// TIA Portal V18 export
FUNCTION_BLOCK "FB_Tower_4Lamp"   // FB5050, LAD
{ S7_Optimized_Access := 'TRUE' }
VERSION : 0.1
// stored: AutoNumber false, IsIECCheckEnabled false, IsRetainMemResEnabled false, MemoryReserve 100, SetENOAutomatically false, UDAEnableTagReadback false
   VAR_INPUT
      iReady : Bool;   // 系统OK
      iManual_Mode : Bool;
      iAuto_Mode : Bool;
      iAuto_Running : Bool;   // 自动运行信号
      iCheck_Mode : Bool;
      iIdle : Bool;   // 自动运行中空闲信号
      iWarning : Bool;
      iFault : Bool;
      "i0.5s_Pulse" : Bool;   // 0.5S脉冲
      i1s_Pulse : Bool;   // 1S脉冲
      i2s_Pulse : Bool;   // 2S脉冲
      iResetButton : Bool;   // 复位按钮
      "iE-StopButtonOK" : Bool;   // 急停按钮未按下
      iSafetyGateClosed : Bool;   // 安全门关闭信号
      iSafetyGateRelayOK : Bool;   // 安全门继电器输出OK
      iPowerOn : Bool;   // 系统上电信号
      iMachineHomePos : Bool;   // 所有设备在原始位
      iWorkAreaLightButton : Bool;   // HMI工作区域照明按钮
      iTest_Lamp : Bool;   // 灯测试按钮
   END_VAR
   VAR_OUTPUT
      oRed_Lamp : Bool;   // 塔灯-红色
      oYellow_Lamp : Bool;   // 塔灯-黄色
      oGreen_Lamp : Bool;   // 塔灯-绿色
      oBlue_Lamp : Bool;   // 塔灯-蓝色 1.蓝灯常亮表示设备在原位;2.蓝灯闪烁表示工位缺料等待上料
      oBuzzer : Bool;   // 塔灯-蜂鸣器
      oPowerOn : Bool;   // 系统上电指示灯
      oResetLamp : Bool;   // 复位按钮指示灯
      oWorkArea1_LightingOn : Bool;   // 工作区域1 照明打开
      oWorkArea2_LightingOn : Bool;   // 工作区域2 照明打开
      oWorkArea3_LightingOn : Bool;   // 工作区域3 照明打开
   END_VAR
   VAR_IN_OUT
      ioStationWaitingLoadPart : Bool;   // 工位等待工位上料
      ioBuzzerON : Bool;   // 蜂鸣器屏蔽开关
      ioBuzzerSetVal : Int;   // 蜂鸣器鸣叫设定值
   END_VAR
   VAR
      TON : Array[0..10] of TON_TIME;
      sRed_Lamp { S7_SetPoint := 'True'} : Bool;
      sResetButtonPressed : Bool;   // 复位按钮已按下
      sBuzzerOnCurrentVal : Int;   // 蜂鸣器鸣叫实际值
      P_TRIG : Array[0..10] of Bool;
      N_TRIG : Array[0..10] of Bool;
   END_VAR
   VAR_TEMP   // added for the SCL form of the ladder/FBD networks
      _w1 : Bool;
      _w2 : Bool;
      _w3 : Bool;
      _w4 : Bool;
      _w5 : Bool;
      _w6 : Bool;
   END_VAR
BEGIN

REGION Network 1: 塔灯-红色 / TowerLamp_Red
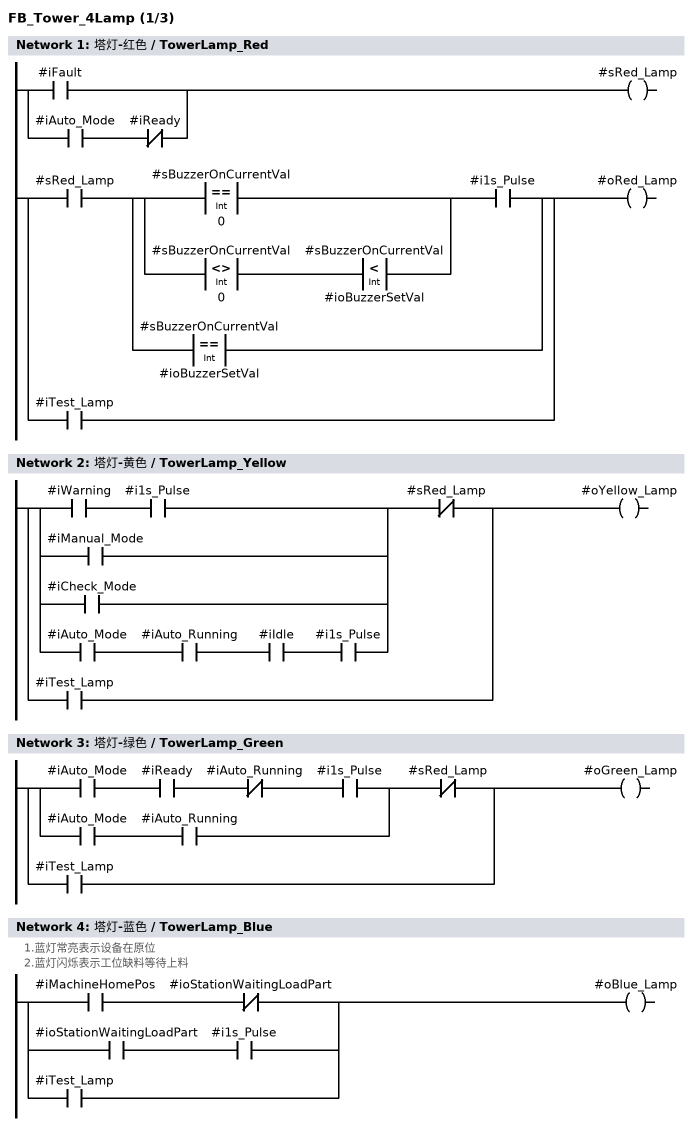
   RUNG wire#powerrail
      Contact( #iFault )
      wire#w1
      Coil( #sRed_Lamp )
   END_RUNG
   RUNG wire#powerrail
      Contact( #iAuto_Mode )
      I_Contact( #iReady )
   END_RUNG wire#w1
   RUNG wire#powerrail
      Contact( #sRed_Lamp )
      wire#w2
      { S7_Templates := "SrcType := Int" } EQ_Contact(in1 := #sBuzzerOnCurrentVal, in2 := 0)
      wire#w3
      Contact( #i1s_Pulse )
      wire#w4
      Coil( #oRed_Lamp )
   END_RUNG
   RUNG wire#w2
      { S7_Templates := "SrcType := Int" } NE_Contact(in1 := #sBuzzerOnCurrentVal, in2 := 0)
      { S7_Templates := "SrcType := Int" } LT_Contact(in1 := #sBuzzerOnCurrentVal, in2 := #ioBuzzerSetVal)
   END_RUNG wire#w3
   RUNG wire#w2
      { S7_Templates := "SrcType := Int" } EQ_Contact(in1 := #sBuzzerOnCurrentVal, in2 := #ioBuzzerSetVal)
   END_RUNG wire#w4
   RUNG wire#powerrail
      Contact( #iTest_Lamp )
   END_RUNG wire#w4
   // the same network as SCL:
   #sRed_Lamp := #iFault OR (#iAuto_Mode AND NOT #iReady);
   #oRed_Lamp := (#sRed_Lamp AND ((((#sBuzzerOnCurrentVal = 0) OR ((#sBuzzerOnCurrentVal <> 0) AND (#sBuzzerOnCurrentVal < #ioBuzzerSetVal))) AND #i1s_Pulse) OR (#sBuzzerOnCurrentVal = #ioBuzzerSetVal))) OR #iTest_Lamp;
END_REGION

REGION Network 2: 塔灯-黄色 / TowerLamp_Yellow
   RUNG wire#powerrail
      Contact( #iWarning )
      Contact( #i1s_Pulse )
      wire#w1
      I_Contact( #sRed_Lamp )
      wire#w2
      Coil( #oYellow_Lamp )
   END_RUNG
   RUNG wire#powerrail
      Contact( #iManual_Mode )
   END_RUNG wire#w1
   RUNG wire#powerrail
      Contact( #iCheck_Mode )
   END_RUNG wire#w1
   RUNG wire#powerrail
      Contact( #iAuto_Mode )
      Contact( #iAuto_Running )
      Contact( #iIdle )
      Contact( #i1s_Pulse )
   END_RUNG wire#w1
   RUNG wire#powerrail
      Contact( #iTest_Lamp )
   END_RUNG wire#w2
   // the same network as SCL:
   #oYellow_Lamp := (((#iWarning AND #i1s_Pulse) OR #iManual_Mode OR #iCheck_Mode OR (#iAuto_Mode AND #iAuto_Running AND #iIdle AND #i1s_Pulse)) AND NOT #sRed_Lamp) OR #iTest_Lamp;
END_REGION

REGION Network 3: 塔灯-绿色 / TowerLamp_Green
   RUNG wire#powerrail
      Contact( #iAuto_Mode )
      Contact( #iReady )
      I_Contact( #iAuto_Running )
      Contact( #i1s_Pulse )
      wire#w1
      I_Contact( #sRed_Lamp )
      wire#w2
      Coil( #oGreen_Lamp )
   END_RUNG
   RUNG wire#powerrail
      Contact( #iAuto_Mode )
      Contact( #iAuto_Running )
   END_RUNG wire#w1
   RUNG wire#powerrail
      Contact( #iTest_Lamp )
   END_RUNG wire#w2
   // the same network as SCL:
   #oGreen_Lamp := (((#iAuto_Mode AND #iReady AND NOT #iAuto_Running AND #i1s_Pulse) OR (#iAuto_Mode AND #iAuto_Running)) AND NOT #sRed_Lamp) OR #iTest_Lamp;
END_REGION

REGION Network 4: 塔灯-蓝色 / TowerLamp_Blue
   // 1.蓝灯常亮表示设备在原位
   // 2.蓝灯闪烁表示工位缺料等待上料
   RUNG wire#powerrail
      Contact( #iMachineHomePos )
      I_Contact( #ioStationWaitingLoadPart )
      wire#w1
      Coil( #oBlue_Lamp )
   END_RUNG
   RUNG wire#powerrail
      Contact( #ioStationWaitingLoadPart )
      Contact( #i1s_Pulse )
   END_RUNG wire#w1
   RUNG wire#powerrail
      Contact( #iTest_Lamp )
   END_RUNG wire#w1
   // the same network as SCL:
   #oBlue_Lamp := (#iMachineHomePos AND NOT #ioStationWaitingLoadPart) OR (#ioStationWaitingLoadPart AND #i1s_Pulse) OR #iTest_Lamp;
END_REGION

REGION Network 5: 蜂鸣器蜂鸣次数 / Number of buzzer buzzes
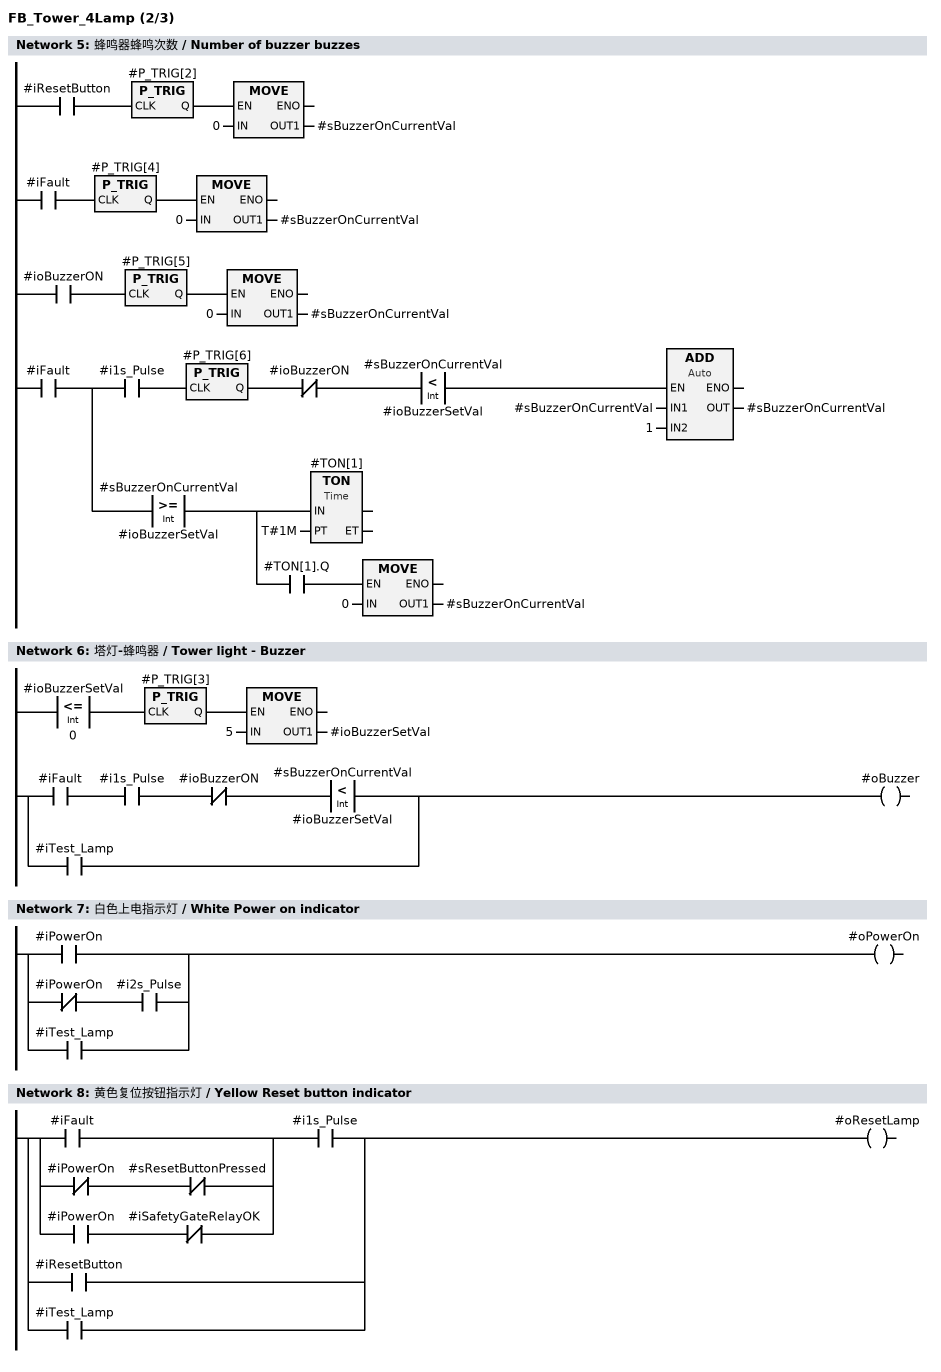
   RUNG wire#powerrail
      Contact( #iResetButton )
      P_Trig( #P_TRIG[2] )
      Move(in := 0, out1 => #sBuzzerOnCurrentVal)
   END_RUNG
   RUNG wire#powerrail
      Contact( #iFault )
      P_Trig( #P_TRIG[4] )
      Move(in := 0, out1 => #sBuzzerOnCurrentVal)
   END_RUNG
   RUNG wire#powerrail
      Contact( #ioBuzzerON )
      P_Trig( #P_TRIG[5] )
      Move(in := 0, out1 => #sBuzzerOnCurrentVal)
   END_RUNG
   RUNG wire#powerrail
      Contact( #iFault )
      wire#w1
      Contact( #i1s_Pulse )
      P_Trig( #P_TRIG[6] )
      I_Contact( #ioBuzzerON )
      { S7_Templates := "SrcType := Int" } LT_Contact(in1 := #sBuzzerOnCurrentVal, in2 := #ioBuzzerSetVal)
      Add(in1 := #sBuzzerOnCurrentVal, in2 := 1, out => #sBuzzerOnCurrentVal)
   END_RUNG
   RUNG wire#w1
      { S7_Templates := "SrcType := Int" } GE_Contact(in1 := #sBuzzerOnCurrentVal, in2 := #ioBuzzerSetVal)
      wire#w2
      { S7_Templates := "time_type := Time" } #TON[1].TON(pt := T#1M, et =>)
   END_RUNG
   RUNG wire#w2
      Contact( #TON[1].Q )
      Move(in := 0, out1 => #sBuzzerOnCurrentVal)
   END_RUNG
   // the same network as SCL:
   #_w1 := #iResetButton AND NOT #P_TRIG[2];   // rising edge
   #P_TRIG[2] := #iResetButton;
   IF #_w1 THEN #sBuzzerOnCurrentVal := 0; END_IF;
   #_w2 := #iFault AND NOT #P_TRIG[4];   // rising edge
   #P_TRIG[4] := #iFault;
   IF #_w2 THEN #sBuzzerOnCurrentVal := 0; END_IF;
   #_w3 := #ioBuzzerON AND NOT #P_TRIG[5];   // rising edge
   #P_TRIG[5] := #ioBuzzerON;
   IF #_w3 THEN #sBuzzerOnCurrentVal := 0; END_IF;
   #_w4 := #iFault AND #i1s_Pulse;
   #_w5 := #_w4 AND NOT #P_TRIG[6];   // rising edge
   #P_TRIG[6] := #_w4;
   IF #_w5 AND NOT #ioBuzzerON AND (#sBuzzerOnCurrentVal < #ioBuzzerSetVal) THEN
       #sBuzzerOnCurrentVal := #sBuzzerOnCurrentVal + 1;
   END_IF;
   #_w6 := #iFault AND (#sBuzzerOnCurrentVal >= #ioBuzzerSetVal);
   #TON[1].TON(IN := #_w6, PT := T#1M);
   IF #_w6 AND #TON[1].Q THEN #sBuzzerOnCurrentVal := 0; END_IF;
END_REGION

REGION Network 6: 塔灯-蜂鸣器 / Tower light - Buzzer
   RUNG wire#powerrail
      { S7_Templates := "SrcType := Int" } LE_Contact(in1 := #ioBuzzerSetVal, in2 := 0)
      P_Trig( #P_TRIG[3] )
      Move(in := 5, out1 => #ioBuzzerSetVal)
   END_RUNG
   RUNG wire#powerrail
      Contact( #iFault )
      Contact( #i1s_Pulse )
      I_Contact( #ioBuzzerON )
      { S7_Templates := "SrcType := Int" } LT_Contact(in1 := #sBuzzerOnCurrentVal, in2 := #ioBuzzerSetVal)
      wire#w1
      Coil( #oBuzzer )
   END_RUNG
   RUNG wire#powerrail
      Contact( #iTest_Lamp )
   END_RUNG wire#w1
   // the same network as SCL:
   #_w1 := #ioBuzzerSetVal <= 0;
   #_w2 := #_w1 AND NOT #P_TRIG[3];   // rising edge
   #P_TRIG[3] := #_w1;
   IF #_w2 THEN #ioBuzzerSetVal := 5; END_IF;
   #oBuzzer := (#iFault AND #i1s_Pulse AND NOT #ioBuzzerON AND (#sBuzzerOnCurrentVal < #ioBuzzerSetVal)) OR #iTest_Lamp;
END_REGION

REGION Network 7: 白色上电指示灯 / White Power on indicator
   RUNG wire#powerrail
      Contact( #iPowerOn )
      wire#w1
      Coil( #oPowerOn )
   END_RUNG
   RUNG wire#powerrail
      I_Contact( #iPowerOn )
      Contact( #i2s_Pulse )
   END_RUNG wire#w1
   RUNG wire#powerrail
      Contact( #iTest_Lamp )
   END_RUNG wire#w1
   // the same network as SCL:
   #oPowerOn := #iPowerOn OR (NOT #iPowerOn AND #i2s_Pulse) OR #iTest_Lamp;
END_REGION

REGION Network 8: 黄色复位按钮指示灯 / Yellow Reset button indicator
   RUNG wire#powerrail
      Contact( #iFault )
      wire#w1
      Contact( #i1s_Pulse )
      wire#w2
      Coil( #oResetLamp )
   END_RUNG
   RUNG wire#powerrail
      I_Contact( #iPowerOn )
      I_Contact( #sResetButtonPressed )
   END_RUNG wire#w1
   RUNG wire#powerrail
      Contact( #iPowerOn )
      I_Contact( #iSafetyGateRelayOK )
   END_RUNG wire#w1
   RUNG wire#powerrail
      Contact( #iResetButton )
   END_RUNG wire#w2
   RUNG wire#powerrail
      Contact( #iTest_Lamp )
   END_RUNG wire#w2
   // the same network as SCL:
   #oResetLamp := ((#iFault OR (NOT #iPowerOn AND NOT #sResetButtonPressed) OR (#iPowerOn AND NOT #iSafetyGateRelayOK)) AND #i1s_Pulse) OR #iResetButton OR #iTest_Lamp;
END_REGION

REGION Network 9: 复位按钮已按下 / The reset button has been pressed
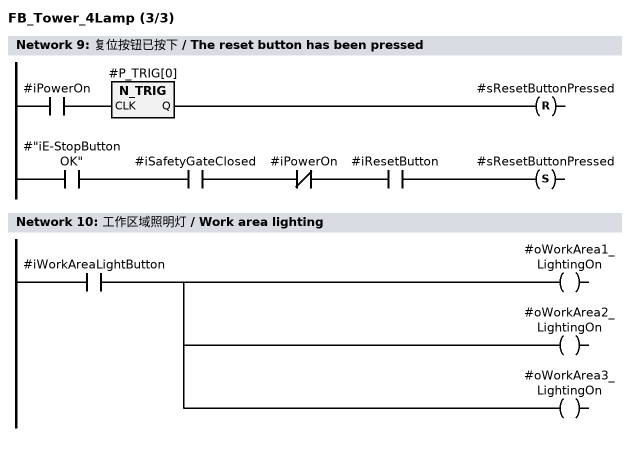
   RUNG wire#powerrail
      Contact( #iPowerOn )
      N_Trig( #P_TRIG[0] )
      R_Coil( #sResetButtonPressed )
   END_RUNG
   RUNG wire#powerrail
      Contact( #"iE-StopButtonOK" )
      Contact( #iSafetyGateClosed )
      I_Contact( #iPowerOn )
      Contact( #iResetButton )
      S_Coil( #sResetButtonPressed )
   END_RUNG
   // the same network as SCL:
   #_w1 := NOT #iPowerOn AND #P_TRIG[0];   // falling edge
   #P_TRIG[0] := #iPowerOn;
   IF #_w1 THEN #sResetButtonPressed := FALSE; END_IF;
   IF #"iE-StopButtonOK" AND #iSafetyGateClosed AND NOT #iPowerOn AND #iResetButton THEN
       #sResetButtonPressed := TRUE;
   END_IF;
END_REGION

REGION Network 10: 工作区域照明灯 / Work area lighting
   RUNG wire#powerrail
      Contact( #iWorkAreaLightButton )
      wire#w1
      Coil( #oWorkArea1_LightingOn )
   END_RUNG
   RUNG wire#w1
      Coil( #oWorkArea2_LightingOn )
   END_RUNG
   RUNG wire#w1
      Coil( #oWorkArea3_LightingOn )
   END_RUNG
   // the same network as SCL:
   #oWorkArea1_LightingOn := #iWorkAreaLightButton;
   #oWorkArea2_LightingOn := #iWorkAreaLightButton;
   #oWorkArea3_LightingOn := #iWorkAreaLightButton;
END_REGION
END_FUNCTION_BLOCK
